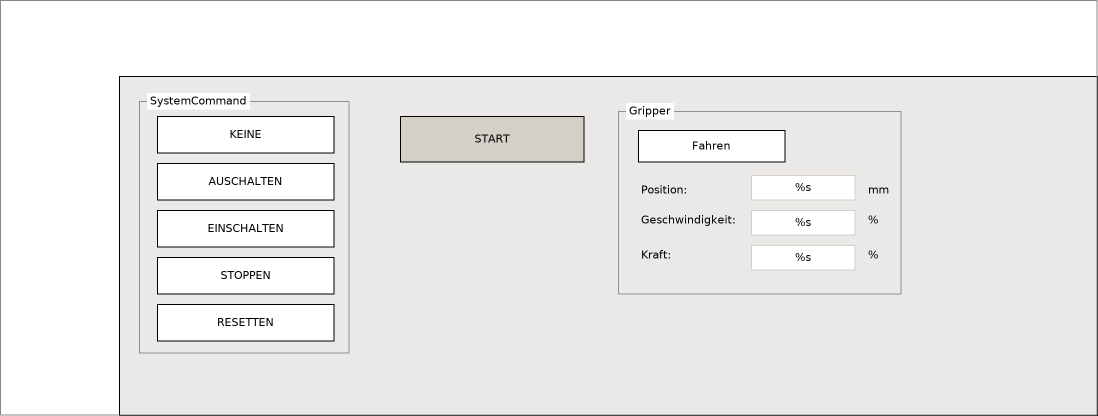
VISUALIZATION Visualization  // 1098x416
VAR_IN_OUT
	
END_VAR

VAR
	iPos		:BYTE;
	iGeschw		:BYTE;
	iKraft		:BYTE;
END_VAR
    Rectangle (119,76 979x340)
    RoundedRectangle (400,116 184x46), "START"
        tap GVL.Execute
    GroupBox (139,93 210x260), "SystemCommand"
        RoundedRectangle (18,70 177x37), "AUSCHALTEN"
            OnMouseClick: execute { GVL.SystemCommand := 1; }
        RoundedRectangle (18,117 177x37), "EINSCHALTEN"
            OnMouseClick: execute { GVL.SystemCommand := 2; }
        RoundedRectangle (18,164 177x37), "STOPPEN"
            OnMouseClick: execute { GVL.SystemCommand := 3; }
        RoundedRectangle (18,211 177x37), "RESETTEN"
            OnMouseClick: execute { GVL.SystemCommand := 4; }
        RoundedRectangle (18,23 177x37), "KEINE"
            OnMouseClick: execute { GVL.SystemCommand := 0; }
    GroupBox (618,103 283x191), "Gripper"
        RoundedRectangle (20,27 147x32), "Fahren"
            OnMouseClick: execute { Anlage.Gripper.A_PositionAnfahren(iPos := iPos, iGeschw := iGeschw, iKraft := iKraft); }
        Textfield (133,72 104x25), "%s", text variable: iPos
            OnMouseDown: write iPos via Edit, format %s
        Textfield (133,107 104x25), "%s", text variable: iGeschw
            OnMouseClick: write iGeschw via Edit, format %d
        Textfield (133,142 104x25), "%s", text variable: iKraft
            OnMouseClick: write iKraft via Edit, format %s
        Label (20,72 95x30), "Position:"
        Label (20,102 95x30), "Geschwindigkeit:"
        Label (20,137 95x30), "Kraft:"
        Label (247,72 30x30), "mm"
        Label (247,102 30x30), "%"
        Label (247,137 25x30), "%"
END_VISUALIZATION

(* stored: Version 1.1.0.1
   Visu Visualization: Id {8ee06d94-1743-4088-a244-af8b854510e9} *)
